Universal Robots PolyScope program: andrea11b.urp

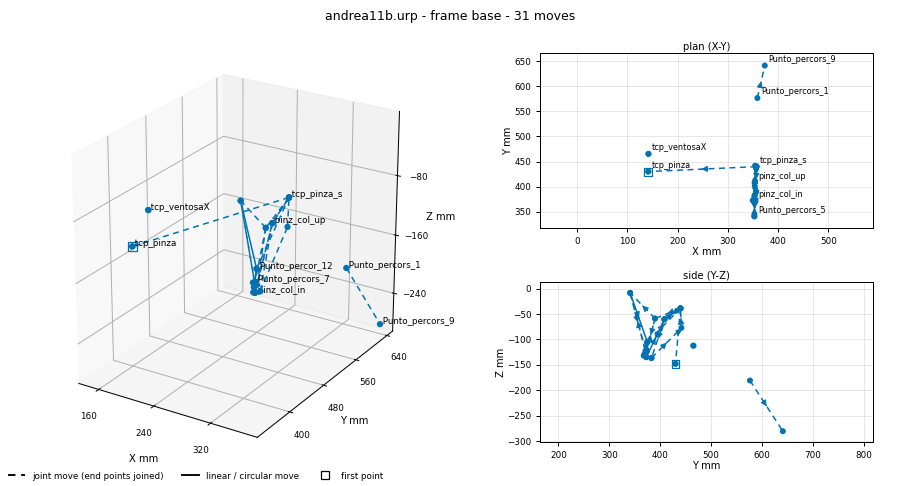
[picture p0: tool path of andrea11b.urp in frame base, 31 of 51 moves have a stored position in this frame; points joined in program order, loops and branches not executed]
Program andrea11b (installation=Kong_install11 directory=/programs/usbdisk/Andrea11b createdIn=3.15.4.106291 lastSavedIn=3.15.4.106291 robotSerialNumber=2017357596)
Calibrated DH parameters: a=[0.000104, -0.381245, -0.385946, 0.00002, 0.000083, 0]; d=[0.089177, 59.99214, -36.297918, -23.584132, 0.094784, 0.082552]; alpha=[1.570197, -0.003145, 0.002952, 1.570494, -1.570091, 0]; deltaTheta=[-0.00001, -0.459739, 0.638868, -0.17972, -0.000006, -0.000462]
InitVariablesNode variables(variable(name=XY, expression=[0,0]), variable(name=ant, expression=3), variable(name=col, expression=4), variable(name=dump, expression=5), variable(name=ghr, expression=2), variable(name=nCycle, expression=0), variable(name=nfc, expression=1), variable(name=pallStocks, expression=[16,16,16,40,16,16,16,40,16,16,16,40,16,40,0,0,0,0,0,0,0,0,0,0]), variable(name=pick, expression=[0,0]))
Robot Program (runOnlyOnce=false)
  Script file /programs/usbdisk/andrea8/nuova dir/relPose.script
    | def relPose(FeaturePose,vect):
    | 
    |     # FeaturePose is the pose for the feature
    |     # vect = p[0.1, 0, 0, 0, 0, 0] makes us move 10cm in the X direction of the feature
    |     # credits: https://forum.universal-robots.com/t/move-tcp-relative-to-feature/15492
    | 
    |    PoseRelativeToFeature = pose_trans(pose_inv(FeaturePose), get_actual_tcp_pose())
    |    MoveTCPRelativeToFeature = pose_add(PoseRelativeToFeature, vect)
    |    return pose_trans(FeaturePose, MoveTCPRelativeToFeature)
    | 
    | end
  Script file /programs/usbdisk/Andrea11b/totf.script
    | def totf(tcpf):
    | 
    |     return sqrt(tcpf[0]*tcpf[0]+tcpf[1]*tcpf[1]+tcpf[2]*tcpf[2]+tcpf[3]*tcpf[3]+tcpf[4]*tcpf[4]+tcpf[5]*tcpf[5])
    | 
    | end
  Script file /programs/usbdisk/andrea8/tcpMov.script
    | def tcpMov(vect):
    | 
    |     # FeaturePose is the pose for the feature
    |     # vect = p[0.1, 0, 0, 0, 0, 0] makes us move 10cm in the X direction of the feature
    |     # credits: https://forum.universal-robots.com/t/move-tcp-relative-to-feature/15492
    | 
    |    tcp_pose = get_actual_tcp_pose()
    |    return pose_add(tcp_pose, vect)
    | 
    | 
    | end
  Script file /home/ur/ursim-current/programs/andrea11/calcItemPosition.script_bak
    | def calcItemPosition(pick, item, pallDefs, grid, featOrigin):
    | 
    |     # calcola la posizione assoluta del pezzo scelto da pickPalletItem
    | 
    |     # nPosX è il numero di colonne
    |     # nPosY è il numero di righe
    |     # distX è la distanza tra colonne
    |     # distY è la distanza tra righe
    |     # [posX1, posY1] è la posizione del primo pezzo rispetto all'origine del pallet
    | 
    |     nPallet = pick[0] + 1 # numero del pallet (gli id partono da 0)
    |     nItem = pick[1] + 1 # numero del pezzo
    | 
    |     nPosXgrid = grid[0] # numero di posizioni della giglia in X
    |     distXgrid = grid[2] # distanza tra gli slot della griglia in X
    |     distYgrid = grid[3] # distanza tra gli slot della griglia in Y
    | 
    |     pallPosX = nPallet%nPosXgrid
    |     if(pallPosX==0): pallPosX = nPosXgrid end
    |     pallPosY = ceil(nPallet/nPosXgrid)
    | 
    |     pallPosX1 = grid[4]
    |     pallPosY1 = grid[5]
    | 
    | 
    |     nPosX = pallDefs[item,0]
    |     nPosY = pallDefs[item,1]
    |     distX = pallDefs[item,2]
    |     distY = pallDefs[item,3]
    |     posX1 = pallDefs[item,4]
    |     posY1 = pallDefs[item,5]
    | 
    |     posX = nItem%nPosX
    |     if(posX==0): posX = nPosX end
    |     posY = ceil(nItem/nPosX)
    | 
    |     # [X,Y] è la posizione del pezzo rispetto all'origine della griglia
    | 
    |     X=distX*(posX - 1) + posX1 + distXgrid*(pallPosX - 1) + pallPosX1
    |     Y=distY*(posY - 1) + posY1 + distYgrid*(pallPosY - 1) + pallPosY1
    |     xy=[X,Y]
    | 
    |     return xy
    | 
    |  end
  Script file /programs/usbdisk/andrea8/pickPalletItem.script
    | def pickPalletItem(type, pallDefs, pallTypes, pallStocks):
    | 
    |   # seleziona un pezzo sulla griglia, noti il tipo di pezzo e lo stato della griglia
    | 
    |   # lo script funziona finché le variabili del robot non vengono resettate. Tuttavia, anche
    |   # in caso di riavvio, è possibile scrivere manualmente le info sulla griglia e lo stock
    |   # all'inizio del programma, così da 'insegnare' al robot dove farlo
    |   # riprendere
    | 
    |   iPallet = 0 # inizializzo l'id del pallet
    | 
    |   while iPallet < length(pallStocks):
    | 
    |     if pallTypes[iPallet] == type and pallStocks[iPallet] > 0 :
    | 
    |       nItems = pallStocks[iPallet] # numero di pezzi nello stock del pallet iesimo
    | 
    |       nPosX = pallDefs[type,0] # numero di posizioni lungo x, come definito per il pallet di tipo "type"
    |       nPosY = pallDefs[type,1] # numero di posizioni lungo y, come definito per il pallet di tipo "type"
    | 
    |       stockMax = nPosX*nPosY
    |       iItem = stockMax - nItems # id del pezzo
    | 
    |       pick = [iPallet,iItem]
    | 
    |       # pick = [id del pallet, id del pezzo]
    | 
    |       return pick
    |  end
    | iPallet = iPallet + 1
    | end
    | end
  Script file /home/ur/ursim-current/programs/andrea11/stockUpdate.script_bak
    | def stockUpdate(pick,stock):
    | 
    |     # simple function that ingests the output of pickItem and returns the
    |     # modified stock array. just so to avoid using global variables and
    |     # multi-dimensional arrays
    | 
    |     i = pick[0]
    |     stock[i] = stock[i] - 1
    |     return stock
    | 
    | 
    | end
  Script file /programs/usbdisk/andrea10/ini_grid.script_bak.script
    | def ini_grid():
    | 
    |     # grid = [nPallPosX, nPallPosY, distPallX, distPallY, pallPosX1, pallPosY1, pallPosZ1]
    |     # la struttura e' del tutto analoga in logica con quella espressa in defs
    |     grid = [4, 4, 90, 90, 10, 20, 6]
    |     return grid
    | end
  Script file /programs/usbdisk/andrea10/ini_defs.script_bak.script
    | def ini_defs():
    | 
    |     # definition = [nPosX,nPosY,distX,distY,posX1,posY1,posZ1]
    | 
    |     # nPosX è il numero di colonne
    |     # nPosY è il numero di righe
    |     # distX è la distanza tra colonne
    |     # distY è la distanza tra righe
    |     # [posX1, posY1] è la posizione del primo pezzo rispetto all'origine del pallet
    |     # posZ1 e' la posizione che deve raggiungere il TCP lungo asse Z, che sarebbe asse verticale
    | 
    |     defs = [
    |         [0, 0, 0, 0, 0, 0, 0], # slot vuoto
    |         [4, 10, 18, 8, 15.5, 3.3, 11.1], # pallet nfc
    |         [4, 4, 21, 21, 16, 11, 49], # pallet ghiere
    |         [1, 1, 0, 0, 132.06, 44, 16.05], # stazione antenna
    |         [1, 2, 0, 40, 20.256, 24, 27.85], # stazione incollaggio
    |         [1, 1, 0, 0, 40, 40, 50] # cestino
    |     ]
    |     return defs
    | end
  Script file /programs/usbdisk/Andrea11b/ini_types.script_bak_bak
    | def ini_types():
    | 
    |     visualTypes = [
    | 
    |         [0, 0, 0, 0],
    |         [0, 0, 0, 0],
    |         [0,0,0,0],
    |         [0,0,0,0],
    |         [0,ghr,0,nfc],
    |         [dump,0,0,0]
    | 
    |     ]
    | 
    | # purtroppo fare questa array vuota di dimensione (righe)x(colonne) per aggirare le limitazioni di UR
    | # bisogna ricordarsi di cambiare questa dichiarazione di types se si cambia dimensione griglia
    | 
    |      types = [0,0,0,0,0,0,0,0,0,0,0,0,0,0,0,0,0,0,0,0,0,0,0,0]
    | 
    |     iii = 0
    |     s = size(visualTypes)
    |     i = 0
    |     while i < s[0]:
    | 
    |         ii=0
    |         while ii < s[1]:
    | 
    |             types[iii] = visualTypes[s[0]-1-i,ii]
    |             ii = ii + 1
    |             iii = iii + 1
    |         end
    |     i = i + 1
    |     end
    |     return types
    | end
  Script file /programs/usbdisk/Andrea11b/ini_stocks2.script
    | def ini_stocks(defs, types):
    | 
    |     global f = -1 # usa questo carattere per inizializzare automaticamente pallet pieni
    | 
    |     visualStocks = [
    | 
    |         [f, f, f, f],
    |         [f, f, f, f],
    |         [f, f, f, f],
    |         [f, f, f, f],
    |         [f, 14, f, f],
    |         [f ,f, f, f]
    | 
    |     ]
    | 
    | # purtroppo fare questa array vuota di dimensione (righe)x(colonne) per aggirare le limitazioni di UR
    | # bisogna ricordarsi di cambiare questa dichiarazione di types se si cambia dimensione griglia
    | 
    |      stocks = [0,0,0,0,0,0,0,0,0,0,0,0,0,0,0,0,0,0,0,0,0,0,0,0]
    | 
    |     iii = 0
    |     s = size(visualStocks)
    |     i = 0
    |     while i < s[0]:
    | 
    |         ii=0
    |         while ii < s[1]:
    |             if visualStocks[s[0]-1-i,ii] == f:
    |                 nPosX = defs[types[iii], 0]
    |                 nPosY = defs[types[iii], 1]
    |                 stocks[iii] = nPosX*nPosY
    |             else:
    | 
    |                 stocks[iii] = visualStocks[s[0]-1-i,ii]
    |             end
    |             ii = ii + 1
    |             iii = iii + 1
    |         end
    |     i = i + 1
    |     end
    |     return stocks
    | end
  Script file /programs/usbdisk/Andrea11b/gen_tcp_grid.script
    | def next_tcp_grid_pos(cur_pos,size,dist):
    | 
    | # size e' la dimensione della griglia da generare,
    | # 2 significa 2x2, 3 significa 3x3 etc
    | 
    | rel_p = [0,0]
    | tcpp = get_actual_tcp_pose()
    | 
    | posX = cur_pos%size
    | if(posX==0): posX = size end
    | posY = ceil(cur_pos/size)
    | 
    | actual_dx = -dist*(size-1)/2 + (posX-1)*dist
    | actual_dy= -dist*(size-1)/2 + (posY-1)*dist
    | 
    | posX = (cur_pos+1)%size
    | if(posX==0): posX = size end
    | posY = ceil((cur_pos+1)/size)
    | 
    | next_dx = -dist*(size-1)/2 + (posX-1)*dist
    | next_dy= -dist*(size-1)/2 + (posY-1)*dist
    | 
    | rel_p = [next_dx - actual_dx, next_dy - actual_dy]
    | 
    | return rel_p
    | 
    | end
  If nCycle≟0
    Set DigitalOutput pin=digital_out[2]; digitalValue=0
    pallTypes := ini_types()
    nfc_ck_override := True
    grid := ini_grid()
    pallDefs := ini_defs()
    pallStocks := ini_stocks(pallDefs,pallTypes)
    SuppressedNode
      Popup Message (haltProgram=false inputType=Variable) variable=grid
    ghr := ghr
    nfc := nfc
    ant := ant
    col := col
    dump := dump
    URCap Close Gripper (SCHUNK End-of-Arm Modular System for UR, SCHUNK GmbH & Co.)
    nCycle := 1
    nfc_check := False
    ghr_check := False
    Wait Sleep waitTime=5
  MoveJ speed 60 deg/s, acceleration 80 deg/s^2 (useActiveTCP=false) tcp=Pinza
    Waypoint tcp_pinza: TCP in base x=141.498 y=430.173 z=-147.715 mm, rx=-2.3787 ry=0.7214 rz=1.7108 rad; joints [-125.948, -50.519, 103.828, -113.29, -23.958, -21.608] deg; pose in feature x=-0.012 y=-0.048 z=150.016 mm, rx=-1.1212 ry=1.1212 rz=0.4102 rad; flange x=182.463 y=570.54 z=26.56 mm, rx=-2.3787 ry=0.7214 rz=1.7108 rad
    item := ghr
    pick := pickPalletItem(item,pallDefs,pallTypes,pallStocks)
    lastpick := pick
    SuppressedNode
      Popup Message (haltProgram=false inputType=Variable) variable=pick
    XY := calcItemPosition(pick, item,pallDefs, grid,piano_moduli)
    p_pall := relPose(piano_moduli,p[XY[0]/1000,XY[1]/1000,0.0,0.0,0.0,0.0])
    SuppressedNode
      Popup Message (haltProgram=false inputType=Variable) variable=XY
    Waypoint Punto_percors (Variable): motionParameters(blendRadius=0.004); variable=p_pall
  MoveL speed 250 mm/s, acceleration 1200 mm/s^2 (useActiveTCP=false) tcp=Pinza; feature=Base
    MoveDirectionNode (selectedDirection=ZMinus toolParams=0.05, 1.2) feature=origine_moduli
      Until DISTANCE (allowActions=true deceleration=3 distanceNodeType=STOP) Distance=0.125; motionParameters(blendRadius=0)
        URCap Open Gripper (SCHUNK End-of-Arm Modular System for UR, SCHUNK GmbH & Co.)
        p_pezzo := relPose(piano_moduli,p[0.0, 0.0, 125/1000, 0.0, 0.0, 0.0])
        Waypoint Punto_percors (Variable): variable=p_pezzo
        pallStocks := stockUpdate(pick,pallStocks)
      Until EXPRESSION (allowActions=true) ExpressionBranch=totf(get_tcp_force())>92
        ghr_check := False
        ghr_attpt := 0
        Loop While (checkContinuously=false) expression=ghr_check≟ False
          SuppressedNode
            MoveL speed 125 mm/s, acceleration 600 mm/s^2 (useActiveTCP=false) tcp=Pinza; feature=Base
              p_pezzo := relPose(piano_moduli,p[0.0, 0.0, -125*0.001, 0.0, 0.0, 0.0])
              Waypoint Punto_percors (Variable): variable=p_pezzo
              URCap Open Gripper (SCHUNK End-of-Arm Modular System for UR, SCHUNK GmbH & Co.)
              p_pezzo := relPose(piano_moduli,p[0.0, 0.0, 125/1000, 0.0, 0.0, 0.0])
              Waypoint Punto_percors (Variable): variable=p_pezzo
              pallStocks := stockUpdate(pick,pallStocks)
              SuppressedNode
                Popup Message (haltProgram=false inputType=Variable) variable=pallStocks
          ghr_attpt := ghr_attpt+1
          MoveL speed 125 mm/s, acceleration 600 mm/s^2 (useActiveTCP=false) tcp=Pinza; feature=Base
            Waypoint Punto_percor_14 (Relative): relativeFromPosition TCP in base x=29.478 y=440.875 z=-307.868 mm, rx=-2.3716 ry=0.6969 rz=1.6945 rad; joints [-115.757, -28.156, 105.846, -162.962, -20.903, 4.096] deg; TCP in base x=29.576 y=447.944 z=-300.79 mm, rx=-2.3716 ry=0.6967 rz=1.6945 rad; joints [-115.45, -28.728, 105.08, -162.418, -20.875, 4.938] deg; flange x=68.514 y=584.323 z=-122.922 mm, rx=-2.3716 ry=0.6967 rz=1.6945 rad
          If ghr_attpt≟4
            ghr_attpt := 0
            MoveL speed 50 mm/s, acceleration 500 mm/s^2 (useActiveTCP=false) tcp=Pinza; feature=Base
              Waypoint Punto_percor_15 (Relative): relativeFromPosition TCP in base x=21.045 y=457.337 z=-272.692 mm, rx=-2.3791 ry=0.7237 rz=1.7113 rad; joints [-114.288, -31.162, 104.237, -160.713, -20.745, 8.28] deg; TCP in base x=23.139 y=462.966 z=-278.334 mm, rx=-2.3791 ry=0.7238 rz=1.7112 rad; joints [-114.249, -30.145, 102.884, -160.48, -20.748, 8.391] deg; flange x=64.258 y=603.606 z=-104.316 mm, rx=-2.3791 ry=0.7238 rz=1.7112 rad
          MoveL speed 50 mm/s, acceleration 500 mm/s^2 (useActiveTCP=false) tcp=Pinza; feature=Base
            Waypoint Punto_percor_10 (Relative): relativeFromPosition TCP in base x=33.913 y=490.369 z=-249.44 mm, rx=-2.3587 ry=0.6534 rz=1.666 rad; joints [-114.038, -33.563, 101.914, -160.666, -20.94, 8.884] deg; TCP in base x=33.89 y=488.921 z=-248.066 mm, rx=-2.3587 ry=0.6535 rz=1.666 rad; joints [-114.091, -33.842, 102.237, -160.564, -20.939, 8.731] deg; flange x=69.127 y=618.113 z=-64.163 mm, rx=-2.3587 ry=0.6535 rz=1.666 rad
          MoveDirectionNode (selectedDirection=ZMinus toolParams=0.05, 1.2) feature=origine_moduli
            Until DISTANCE (allowActions=true deceleration=3 distanceNodeType=STOP) Distance=0.018; motionParameters(blendRadius=0)
              URCap Open Gripper (SCHUNK End-of-Arm Modular System for UR, SCHUNK GmbH & Co.)
              p_pezzo := relPose(piano_moduli,p[0.0, 0.0, 125/1000, 0.0, 0.0, 0.0])
              Waypoint Punto_percors (Variable): variable=p_pezzo
              pallStocks := stockUpdate(pick,pallStocks)
              ghr_check := True
            Until EXPRESSION (allowActions=true) ExpressionBranch=totf(get_tcp_force())>85
              MoveL speed 50 mm/s, acceleration 500 mm/s^2 (useActiveTCP=true) feature=Base
                Waypoint Punto_percors_6 (Relative): relativeFromPosition TCP in base x=4.07 y=674.667 z=69.754 mm, rx=1.9149 ry=-1.1485 rz=-1.8457 rad; joints [-112.275, -36.345, 91.167, -133.706, -10.047, 30.658] deg; TCP in base x=4.143 y=678.166 z=73.281 mm, rx=1.9147 ry=-1.1486 rz=-1.8457 rad; joints [-112.167, -36.367, 90.585, -133.706, -10.021, 31.279] deg; flange x=70.38 y=685.456 z=-8.016 mm, rx=1.9147 ry=-1.1486 rz=-1.8457 rad
  nfc_check := False
  Loop While (checkContinuously=false) expression=nfc_check≟ False
    MoveJ speed 60 deg/s, acceleration 80 deg/s^2 (useActiveTCP=false) tcp=Ventosa
      Waypoint tcp_ventosaX: TCP in base x=141.953 y=465.356 z=-112.213 mm, rx=-2.2886 ry=-0.6046 rz=-0.263 rad; joints [-121.609, -49.485, 100.63, -2.12, 68.781, 127.146] deg; flange x=141.931 y=500.256 z=-13.059 mm, rx=-2.2886 ry=-0.6046 rz=-0.263 rad
      item := dump
      pick := pickPalletItem(item,pallDefs,pallTypes,pallStocks)
      SuppressedNode
        Popup Message (haltProgram=false inputType=Variable) variable=pick
      XY := calcItemPosition(pick, item,pallDefs, grid,piano_moduli)
      p_pall := relPose(piano_moduli,p[XY[0]/1000,XY[1]/1000,0.0,0.0,0.0,0.0])
      SuppressedNode
        Popup Message (haltProgram=false inputType=Variable) variable=XY
      Waypoint Punto_percors (Variable): motionParameters(blendRadius=0.005); variable=p_pall
      Set DigitalOutput pin=digital_out[2]; digitalValue=0
    MoveJ speed 60 deg/s, acceleration 80 deg/s^2 (useActiveTCP=false) tcp=Ventosa
      Waypoint tcp_ventosaX: TCP in base x=141.953 y=465.356 z=-112.213 mm, rx=-2.2886 ry=-0.6046 rz=-0.263 rad; joints [-121.609, -49.485, 100.63, -2.12, 68.781, 127.146] deg; flange x=141.931 y=500.256 z=-13.059 mm, rx=-2.2886 ry=-0.6046 rz=-0.263 rad
      SuppressedNode
        Waypoint tcp_ventosaY_s: TCP in base x=355.984 y=389.916 z=-58.857 mm, rx=-1.401 ry=-1.0647 rz=1.3858 rad; joints [-146.472, -36.177, 73.345, -37.097, -55.375, 194.745] deg; pose in feature x=141.985 y=465.345 z=-112.215 mm, rx=-1.4011 ry=-1.0646 rz=1.3857 rad; flange x=401.93 y=456.119 z=8.64 mm, rx=-1.401 ry=-1.0647 rz=1.3858 rad
      item := nfc
      pick := pickPalletItem(item,pallDefs,pallTypes,pallStocks)
      SuppressedNode
        Popup Message (haltProgram=false inputType=Variable) variable=pick
      XY := calcItemPosition(pick, item,pallDefs, grid,piano_moduli)
      p_pall := relPose(piano_moduli,p[XY[0]/1000,XY[1]/1000,0.0,0.0,0.0,0.0])
      SuppressedNode
        Popup Message (haltProgram=false inputType=Variable) variable=XY
      Waypoint Punto_percors (Variable): motionParameters(blendRadius=0.005); variable=p_pall
    MoveL speed 250 mm/s, acceleration 1200 mm/s^2 (useActiveTCP=false) tcp=Ventosa; feature=Base
      p_pezzo := relPose(piano_moduli,p[0.0, 0.0, -183*0.001, 0.0, 0.0, 0.0])
      Waypoint Punto_percors (Variable): variable=p_pezzo
      Set DigitalOutput pin=digital_out[2]; digitalValue=1
      Wait Sleep waitTime=2
      p_pezzo := relPose(piano_moduli,p[0.0, 0.0, 183/1000, 0.0, 0.0, 0.0])
      Waypoint Punto_percors (Variable): variable=p_pezzo
      pallStocks := stockUpdate(pick,pallStocks)
      SuppressedNode
        Popup Message (haltProgram=false inputType=Variable) variable=pallStocks
    MoveJ speed 60 deg/s, acceleration 80 deg/s^2 (useActiveTCP=false) tcp=Ventosa
      Waypoint Punto_percors_1: motionParameters(blendRadius=0.005); TCP in base x=358.691 y=576.543 z=-180.701 mm, rx=-2.2887 ry=-0.6045 rz=-0.2628 rad; joints [-132.678, -21.575, 54.335, 20.288, 61.783, 117.598] deg; flange x=358.684 y=611.454 z=-81.55 mm, rx=-2.2887 ry=-0.6045 rz=-0.2628 rad
      Waypoint Punto_percors_9: TCP in base x=373.401 y=641.171 z=-280.298 mm, rx=-2.2781 ry=-0.6996 rz=-0.1741 rad; joints [-130.196, 7.244, 8.465, 40.912, 59.771, 115.067] deg; flange x=373.185 y=678.65 z=-182.089 mm, rx=-2.2781 ry=-0.6996 rz=-0.1741 rad
    MoveL speed 250 mm/s, acceleration 1200 mm/s^2 (useActiveTCP=false) tcp=Ventosa; feature=Base
      p_pezzo := relPose(piano_moduli,p[0.0, 0.0, -67*0.001, 0.0, 0.0, 0.0])
      Waypoint Punto_percors (Variable): variable=p_pezzo
      SuppressedNode
        Wait Sleep waitTime=2.5
      If nfc_ck_override≟ True
        nfc_check := True
      Loop Counting (count=5) loopVariable(name=Ciclo_2)
        Wait Sleep waitTime=0.5
        If digital_in[4]≟ True
          nfc_check := True
      p_pezzo := relPose(piano_moduli,p[0.0, 0.0, 70/1000, 0.0, 0.0, 0.0])
      Waypoint Punto_percors (Variable): variable=p_pezzo
  MoveJ speed 60 deg/s, acceleration 80 deg/s^2 (useActiveTCP=false) tcp=Pinza
    Waypoint tcp_pinza_s: TCP in base x=356.783 y=439.979 z=-38.857 mm, rx=1.9379 ry=-1.1643 rz=-1.0823 rad; joints [-132.207, -20.407, 45.734, -60.67, -53.979, 1] deg; flange x=387.119 y=665.322 z=-46.123 mm, rx=1.9379 ry=-1.1643 rz=-1.0823 rad
    Waypoint pinz_col_up: TCP in base x=353.537 y=408.471 z=-60.29 mm, rx=1.9378 ry=-1.1643 rz=-1.0825 rad; joints [-133.591, -22.853, 54.464, -66.388, -55.09, 0.038] deg; flange x=383.886 y=633.812 z=-67.559 mm, rx=1.9378 ry=-1.1643 rz=-1.0825 rad
    Waypoint pinz_col_in: TCP in base x=352.248 y=372.767 z=-134.879 mm, rx=1.8715 ry=-1.2053 rz=-0.9224 rad; joints [-134.79, -16.6, 58.956, -76.087, -61.476, 5.632] deg; flange x=378.139 y=595.635 z=-172.455 mm, rx=1.8715 ry=-1.2053 rz=-0.9224 rad
    URCap Close Gripper (SCHUNK End-of-Arm Modular System for UR, SCHUNK GmbH & Co.)
    Waypoint pinz_col_out: TCP in base x=353.252 y=383.01 z=-136.492 mm, rx=1.8482 ry=-1.2116 rz=-0.904 rad; joints [-134.313, -14.601, 55.679, -74.213, -61.596, 6.906] deg; flange x=379.232 y=604.751 z=-180.176 mm, rx=1.8482 ry=-1.2116 rz=-0.904 rad
    SuppressedNode
      Waypoint pinz_col_up: TCP in base x=353.537 y=408.471 z=-60.29 mm, rx=1.9378 ry=-1.1643 rz=-1.0825 rad; joints [-133.591, -22.853, 54.464, -66.388, -55.09, 0.038] deg; flange x=383.886 y=633.812 z=-67.559 mm, rx=1.9378 ry=-1.1643 rz=-1.0825 rad
    Waypoint Punto_percors_2: TCP in base x=354.064 y=441.822 z=-77.166 mm, rx=1.8482 ry=-1.2116 rz=-0.904 rad; joints [-131.419, -13.619, 42.947, -63.355, -59.194, 8.709] deg; flange x=380.052 y=663.563 z=-120.852 mm, rx=1.8482 ry=-1.2116 rz=-0.904 rad
    SuppressedNode
      URCap Open Gripper (SCHUNK End-of-Arm Modular System for UR, SCHUNK GmbH & Co.)
    Waypoint tcp_pinza_s: TCP in base x=356.783 y=439.979 z=-38.857 mm, rx=1.9379 ry=-1.1643 rz=-1.0823 rad; joints [-132.207, -20.407, 45.734, -60.67, -53.979, 1] deg; flange x=387.119 y=665.322 z=-46.123 mm, rx=1.9379 ry=-1.1643 rz=-1.0823 rad
  MoveJ speed 60 deg/s, acceleration 80 deg/s^2 (useActiveTCP=false) tcp=Dosatore_Colla
    Waypoint tcp_coll_s: TCP in base x=355.98 y=389.944 z=-58.821 mm, rx=-0.0221 ry=-3.1138 rz=0.4025 rad; joints [-139.161, -64.308, 106.34, -121.985, -100.827, 102.96] deg; flange x=356.624 y=435.245 z=113.503 mm, rx=0.7684 ry=-2.9515 rz=0.3801 rad
    Waypoint Punto_percors_7: motionParameters(blendRadius=0); TCP in base x=351.74 y=373.802 z=-121.516 mm, rx=-0.022 ry=-3.1139 rz=0.4024 rad; joints [-140.141, -59.264, 111.047, -131.929, -101.033, 101.993] deg; flange x=352.361 y=419.041 z=50.638 mm, rx=0.7686 ry=-2.9516 rz=0.38 rad
    Waypoint Punto_percors_8: motionParameters(blendRadius=0); TCP in base x=351.721 y=371.153 z=-127.085 mm, rx=-0.022 ry=-3.1138 rz=0.4026 rad; joints [-140.348, -58.803, 111.513, -132.884, -101.078, 101.787] deg; flange x=352.351 y=416.425 z=45.06 mm, rx=0.7686 ry=-2.9515 rz=0.3802 rad
    Waypoint Punto_percors_7: motionParameters(blendRadius=0); TCP in base x=351.74 y=373.802 z=-121.516 mm, rx=-0.022 ry=-3.1139 rz=0.4024 rad; joints [-140.141, -59.264, 111.047, -131.929, -101.033, 101.993] deg; flange x=352.361 y=419.041 z=50.638 mm, rx=0.7686 ry=-2.9516 rz=0.38 rad
    SuppressedNode
      Waypoint tcp_colla: TCP in base x=141.953 y=465.356 z=-112.213 mm, rx=-0.0207 ry=-2.9002 rz=1.1933 rad; joints [-112.251, -46.475, 88.048, -88.757, -104.681, 134.691] deg; flange x=143.75 y=590.738 z=14.373 mm, rx=0.6882 ry=-2.6438 rz=1.0836 rad
  MoveL speed 250 mm/s, acceleration 1200 mm/s^2 (useActiveTCP=false) tcp=Dosatore_Colla; feature=Base
    Waypoint arco01: TCP in base x=349.484 y=372.821 z=-122.517 mm, rx=-0.3054 ry=2.8059 rz=-0.3653 rad; joints [-134.698, -59.864, 121.564, -155.634, -112.071, 92.496] deg; flange x=293.567 y=411.329 z=42.026 mm, rx=-1.0435 ry=2.6885 rz=-0.4726 rad
    Wait Sleep waitTime=0.1
    Waypoint Punto_percors_3: TCP in base x=354.975 y=372.908 z=-124.117 mm, rx=-0.4267 ry=-2.7025 rz=0.3458 rad; joints [-148.003, -53.452, 98.947, -109.424, -86.246, 109.428] deg; flange x=426.96 y=404.747 z=35.534 mm, rx=0.2834 ry=-2.6841 rz=0.1927 rad
  MoveJ speed 60 deg/s, acceleration 80 deg/s^2 (useActiveTCP=false) tcp=Dosatore_Colla
    Waypoint tcp_coll_s: motionParameters(blendRadius=0.005); TCP in base x=355.98 y=389.944 z=-58.821 mm, rx=-0.0221 ry=-3.1138 rz=0.4025 rad; joints [-139.161, -64.308, 106.34, -121.985, -100.827, 102.96] deg; flange x=356.624 y=435.245 z=113.503 mm, rx=0.7684 ry=-2.9515 rz=0.3801 rad
  MoveJ speed 60 deg/s, acceleration 80 deg/s^2 (useActiveTCP=false) tcp=Ventosa
    SuppressedNode
      Waypoint tcp_ventosaY_s: TCP in base x=355.984 y=389.916 z=-58.857 mm, rx=-1.401 ry=-1.0647 rz=1.3858 rad; joints [-146.472, -36.177, 73.345, -37.097, -55.375, 194.745] deg; flange x=401.93 y=456.119 z=8.64 mm, rx=-1.401 ry=-1.0647 rz=1.3858 rad
    Waypoint Punto_percors_5: TCP in base x=352.704 y=341.071 z=-8.564 mm, rx=-1.0185 ry=-1.3146 rz=1.0001 rad; joints [-153.565, -49.242, 85.748, -36.404, -62.461, 164.703] deg; flange x=398.057 y=364.583 z=83.305 mm, rx=-1.0185 ry=-1.3146 rz=1.0001 rad
    Waypoint Punto_percor_11: TCP in base x=353.128 y=371.062 z=-122.13 mm, rx=-1.0185 ry=-1.3145 rz=1.0002 rad; joints [-151.072, -37.136, 83.027, -45.814, -59.963, 164.771] deg; flange x=398.49 y=394.587 z=-30.269 mm, rx=-1.0185 ry=-1.3145 rz=1.0002 rad
    Wait Sleep waitTime=1
    Set DigitalOutput pin=digital_out[2]; digitalValue=0
    Wait Sleep waitTime=1
    Waypoint Punto_percors_5: TCP in base x=352.704 y=341.071 z=-8.564 mm, rx=-1.0185 ry=-1.3146 rz=1.0001 rad; joints [-153.565, -49.242, 85.748, -36.404, -62.461, 164.703] deg; flange x=398.057 y=364.583 z=83.305 mm, rx=-1.0185 ry=-1.3146 rz=1.0001 rad
    SuppressedNode
      Waypoint Punto_percors_4: 
  MoveL speed 250 mm/s, acceleration 1200 mm/s^2 (useActiveTCP=false) tcp=Pressa; feature=Base
    Waypoint Punto_percor_12: motionParameters(blendRadius=0.005); TCP in base x=353.182 y=374.819 z=-104.948 mm, rx=0.1982 ry=-1.5625 rz=-0.2204 rad; joints [-149.346, -43.269, 79.423, -36.069, -58.24, 74.726] deg; flange x=398.78 y=416.125 z=54.625 mm, rx=0.1982 ry=-1.5625 rz=-0.2204 rad
    Waypoint Punto_percor_13: TCP in base x=353.081 y=367.784 z=-131.982 mm, rx=0.1982 ry=-1.5627 rz=-0.2205 rad; joints [-149.903, -41.525, 80.906, -39.318, -58.787, 74.74] deg; flange x=398.651 y=409.066 z=27.605 mm, rx=0.1982 ry=-1.5627 rz=-0.2205 rad
    Wait Sleep waitTime=2
    Waypoint Punto_percor_12: TCP in base x=353.182 y=374.819 z=-104.948 mm, rx=0.1982 ry=-1.5625 rz=-0.2204 rad; joints [-149.346, -43.269, 79.423, -36.069, -58.24, 74.726] deg; flange x=398.78 y=416.125 z=54.625 mm, rx=0.1982 ry=-1.5625 rz=-0.2204 rad
    SuppressedNode
      Waypoint tcp_pressaY: TCP in base x=141.469 y=430.16 z=-147.709 mm, rx=-0.2128 ry=-1.5595 rz=0.1907 rad; joints [-127.014, -38.383, 85.876, -47.443, -35.896, 104.766] deg; flange x=188.109 y=545.63 z=-30.49 mm, rx=-0.2128 ry=-1.5595 rz=0.1907 rad
    SuppressedNode
      Waypoint tcp_pressaX: TCP in base x=141.415 y=430.194 z=-147.729 mm, rx=-1.3127 ry=-2.237 rz=-0.9404 rad; joints [-120.759, -49.8, 97.992, 0.536, 69.418, 38.219] deg; flange x=142.623 y=514.321 z=1.167 mm, rx=-1.3127 ry=-2.237 rz=-0.9404 rad
  MoveJ speed 60 deg/s, acceleration 80 deg/s^2 (useActiveTCP=false) tcp=Pinza
    Waypoint tcp_pinza_s: TCP in base x=356.783 y=439.979 z=-38.857 mm, rx=1.9379 ry=-1.1643 rz=-1.0823 rad; joints [-132.207, -20.407, 45.734, -60.67, -53.979, 1] deg; flange x=387.119 y=665.322 z=-46.123 mm, rx=1.9379 ry=-1.1643 rz=-1.0823 rad
    Waypoint pinz_col_up: TCP in base x=353.537 y=408.471 z=-60.29 mm, rx=1.9378 ry=-1.1643 rz=-1.0825 rad; joints [-133.591, -22.853, 54.464, -66.388, -55.09, 0.038] deg; flange x=383.886 y=633.812 z=-67.559 mm, rx=1.9378 ry=-1.1643 rz=-1.0825 rad
    Waypoint pinz_col_out: TCP in base x=353.252 y=383.01 z=-136.492 mm, rx=1.8482 ry=-1.2116 rz=-0.904 rad; joints [-134.313, -14.601, 55.679, -74.213, -61.596, 6.906] deg; flange x=379.232 y=604.751 z=-180.176 mm, rx=1.8482 ry=-1.2116 rz=-0.904 rad
    Waypoint pinz_col_in: TCP in base x=352.248 y=372.767 z=-134.879 mm, rx=1.8715 ry=-1.2053 rz=-0.9224 rad; joints [-134.79, -16.6, 58.956, -76.087, -61.476, 5.632] deg; flange x=378.139 y=595.635 z=-172.455 mm, rx=1.8715 ry=-1.2053 rz=-0.9224 rad
    URCap Open Gripper (SCHUNK End-of-Arm Modular System for UR, SCHUNK GmbH & Co.)
    Waypoint pinz_col_up: TCP in base x=353.537 y=408.471 z=-60.29 mm, rx=1.9378 ry=-1.1643 rz=-1.0825 rad; joints [-133.591, -22.853, 54.464, -66.388, -55.09, 0.038] deg; flange x=383.886 y=633.812 z=-67.559 mm, rx=1.9378 ry=-1.1643 rz=-1.0825 rad
    SuppressedNode
      Waypoint pinz_col_up: TCP in base x=353.537 y=408.471 z=-60.29 mm, rx=1.9378 ry=-1.1643 rz=-1.0825 rad; joints [-133.591, -22.853, 54.464, -66.388, -55.09, 0.038] deg; flange x=383.886 y=633.812 z=-67.559 mm, rx=1.9378 ry=-1.1643 rz=-1.0825 rad
    SuppressedNode
      Waypoint Punto_percors_2: TCP in base x=354.064 y=441.822 z=-77.166 mm, rx=1.8482 ry=-1.2116 rz=-0.904 rad; joints [-131.419, -13.619, 42.947, -63.355, -59.194, 8.709] deg; flange x=380.052 y=663.563 z=-120.852 mm, rx=1.8482 ry=-1.2116 rz=-0.904 rad
    SuppressedNode
      URCap Open Gripper (SCHUNK End-of-Arm Modular System for UR, SCHUNK GmbH & Co.)
    Waypoint tcp_pinza_s: TCP in base x=356.783 y=439.979 z=-38.857 mm, rx=1.9379 ry=-1.1643 rz=-1.0823 rad; joints [-132.207, -20.407, 45.734, -60.67, -53.979, 1] deg; flange x=387.119 y=665.322 z=-46.123 mm, rx=1.9379 ry=-1.1643 rz=-1.0823 rad
  MoveJ speed 60 deg/s, acceleration 80 deg/s^2 (useActiveTCP=false) tcp=Pinza
    Waypoint tcp_pinza: TCP in base x=141.498 y=430.173 z=-147.715 mm, rx=-2.3787 ry=0.7214 rz=1.7108 rad; joints [-125.948, -50.519, 103.828, -113.29, -23.958, -21.608] deg; pose in feature x=-0.012 y=-0.048 z=150.016 mm, rx=-1.1212 ry=1.1212 rz=0.4102 rad; flange x=182.463 y=570.54 z=26.56 mm, rx=-2.3787 ry=0.7214 rz=1.7108 rad
    SuppressedNode
      Popup Message (haltProgram=false inputType=Variable) variable=pick
    XY := calcItemPosition(lastpick, item,pallDefs, grid,piano_moduli)
    p_pall := relPose(piano_moduli,p[XY[0]/1000-0.000,XY[1]/1000-0.0035,0.0,0.0,0.0,0.0])
    SuppressedNode
      Popup Message (haltProgram=false inputType=Variable) variable=XY
    Waypoint Punto_percors (Variable): motionParameters(blendRadius=0.004); variable=p_pall
  MoveL speed 250 mm/s, acceleration 1200 mm/s^2 (useActiveTCP=false) tcp=Pinza; feature=Base
    MoveDirectionNode (selectedDirection=ZMinus toolParams=0.05, 1.2) feature=origine_moduli
      Until DISTANCE (allowActions=true deceleration=3 distanceNodeType=STOP) Distance=0.11; motionParameters(blendRadius=0)
        URCap Close Gripper (SCHUNK End-of-Arm Modular System for UR, SCHUNK GmbH & Co.)
        p_pezzo := relPose(piano_moduli,p[0.0, 0.0, 125/1000, 0.0, 0.0, 0.0])
        Waypoint Punto_percors (Variable): variable=p_pezzo
        pallStocks := stockUpdate(pick,pallStocks)
      Until EXPRESSION (allowActions=true) ExpressionBranch=totf(get_tcp_force())>95
        ghr_check := False
        ghr_attpt := 0
        Loop While (checkContinuously=false) expression=ghr_check≟ False
          SuppressedNode
            MoveL speed 125 mm/s, acceleration 600 mm/s^2 (useActiveTCP=false) tcp=Pinza; feature=Base
              p_pezzo := relPose(piano_moduli,p[0.0, 0.0, -125*0.001, 0.0, 0.0, 0.0])
              Waypoint Punto_percors (Variable): variable=p_pezzo
              URCap Open Gripper (SCHUNK End-of-Arm Modular System for UR, SCHUNK GmbH & Co.)
              p_pezzo := relPose(piano_moduli,p[0.0, 0.0, 125/1000, 0.0, 0.0, 0.0])
              Waypoint Punto_percors (Variable): variable=p_pezzo
              pallStocks := stockUpdate(pick,pallStocks)
              SuppressedNode
                Popup Message (haltProgram=false inputType=Variable) variable=pallStocks
          ghr_attpt := ghr_attpt+1
          MoveL speed 125 mm/s, acceleration 600 mm/s^2 (useActiveTCP=false) tcp=Pinza; feature=Base
            Waypoint Punto_percor_16 (Relative): relativeFromPosition TCP in base x=21.48 y=497.646 z=-275.999 mm, rx=-2.3783 ry=0.7214 rz=1.7109 rad; joints [-112.781, -28.123, 96.79, -160.334, -20.71, 12.471] deg; TCP in base x=21.716 y=511.71 z=-261.76 mm, rx=-2.3784 ry=0.7216 rz=1.7108 rad; joints [-112.302, -28.904, 94.899, -158.934, -20.726, 13.834] deg; flange x=62.735 y=652.049 z=-87.475 mm, rx=-2.3784 ry=0.7216 rz=1.7108 rad
          If ghr_attpt≟4
            ghr_attpt := 1
            MoveL speed 50 mm/s, acceleration 500 mm/s^2 (useActiveTCP=false) tcp=Pinza; feature=Base
              Waypoint Punto_percor_15 (Relative): relativeFromPosition TCP in base x=21.045 y=457.337 z=-272.692 mm, rx=-2.3791 ry=0.7237 rz=1.7113 rad; joints [-114.288, -31.162, 104.237, -160.713, -20.745, 8.28] deg; TCP in base x=23.139 y=462.966 z=-278.334 mm, rx=-2.3791 ry=0.7238 rz=1.7112 rad; joints [-114.249, -30.145, 102.884, -160.48, -20.748, 8.391] deg; flange x=64.258 y=603.606 z=-104.316 mm, rx=-2.3791 ry=0.7238 rz=1.7112 rad
          MoveL speed 50 mm/s, acceleration 500 mm/s^2 (useActiveTCP=false) tcp=Pinza; feature=Base
            Waypoint Punto_percor_10 (Relative): relativeFromPosition TCP in base x=33.913 y=490.369 z=-249.44 mm, rx=-2.3587 ry=0.6534 rz=1.666 rad; joints [-114.038, -33.563, 101.914, -160.666, -20.94, 8.884] deg; TCP in base x=33.89 y=488.921 z=-248.066 mm, rx=-2.3587 ry=0.6535 rz=1.666 rad; joints [-114.091, -33.842, 102.237, -160.564, -20.939, 8.731] deg; flange x=69.127 y=618.113 z=-64.163 mm, rx=-2.3587 ry=0.6535 rz=1.666 rad
          MoveDirectionNode (selectedDirection=ZMinus toolParams=0.05, 1.2) feature=origine_moduli
            Until DISTANCE (allowActions=true deceleration=3 distanceNodeType=STOP) Distance=0.02; motionParameters(blendRadius=0)
              URCap Close Gripper (SCHUNK End-of-Arm Modular System for UR, SCHUNK GmbH & Co.)
              p_pezzo := relPose(piano_moduli,p[0.0, 0.0, 125/1000, 0.0, 0.0, 0.0])
              Waypoint Punto_percors (Variable): variable=p_pezzo
              pallStocks := stockUpdate(pick,pallStocks)
              ghr_check := True
            Until EXPRESSION (allowActions=true) ExpressionBranch=totf(get_tcp_force())>85
              MoveL speed 50 mm/s, acceleration 500 mm/s^2 (useActiveTCP=true) feature=Base
                Waypoint Punto_percors_6 (Relative): relativeFromPosition TCP in base x=4.07 y=674.667 z=69.754 mm, rx=1.9149 ry=-1.1485 rz=-1.8457 rad; joints [-112.275, -36.345, 91.167, -133.706, -10.047, 30.658] deg; TCP in base x=4.143 y=678.166 z=73.281 mm, rx=1.9147 ry=-1.1486 rz=-1.8457 rad; joints [-112.167, -36.367, 90.585, -133.706, -10.021, 31.279] deg; flange x=70.38 y=685.456 z=-8.016 mm, rx=1.9147 ry=-1.1486 rz=-1.8457 rad
  SuppressedNode
    Popup Message (haltProgram=false inputType=Variable) variable=pick
